# EPICS autosave request: iocBoot/iocHindsXray/auto_positions.req
file "CARS_8_motor_positions.req", P=$(P)
